FUNCTION_BLOCK NOT_DWORD (* IEC 61131-3 Bitwise NOT *)
  (* Standard: 61131-3 *)
  (* Version 0.0, 2004-12-15, JHC, Rockwell Automation, Converted from SRC format. *)
  (* Compiler header: package fb.rt.plc.bits; *)
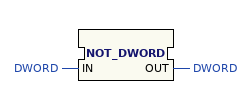
  VAR_INPUT
    IN : DWORD;
  END_VAR
  VAR_OUTPUT
    OUT : DWORD;
  END_VAR
END_FUNCTION_BLOCK
